// TIA Portal V20 export
FUNCTION_BLOCK "LER_Vision_XGX2000_Conversion"   // FB109, LAD
// stored: Access Published, MemoryReserve 100, SetENOAutomatically false
   VAR_INPUT
      VisionData : "LER_typeVisionMonitoring";
   END_VAR
   VAR_OUTPUT
      VisionDataConvert : "LER_typeVisionResultData";
   END_VAR
BEGIN

REGION Network 1
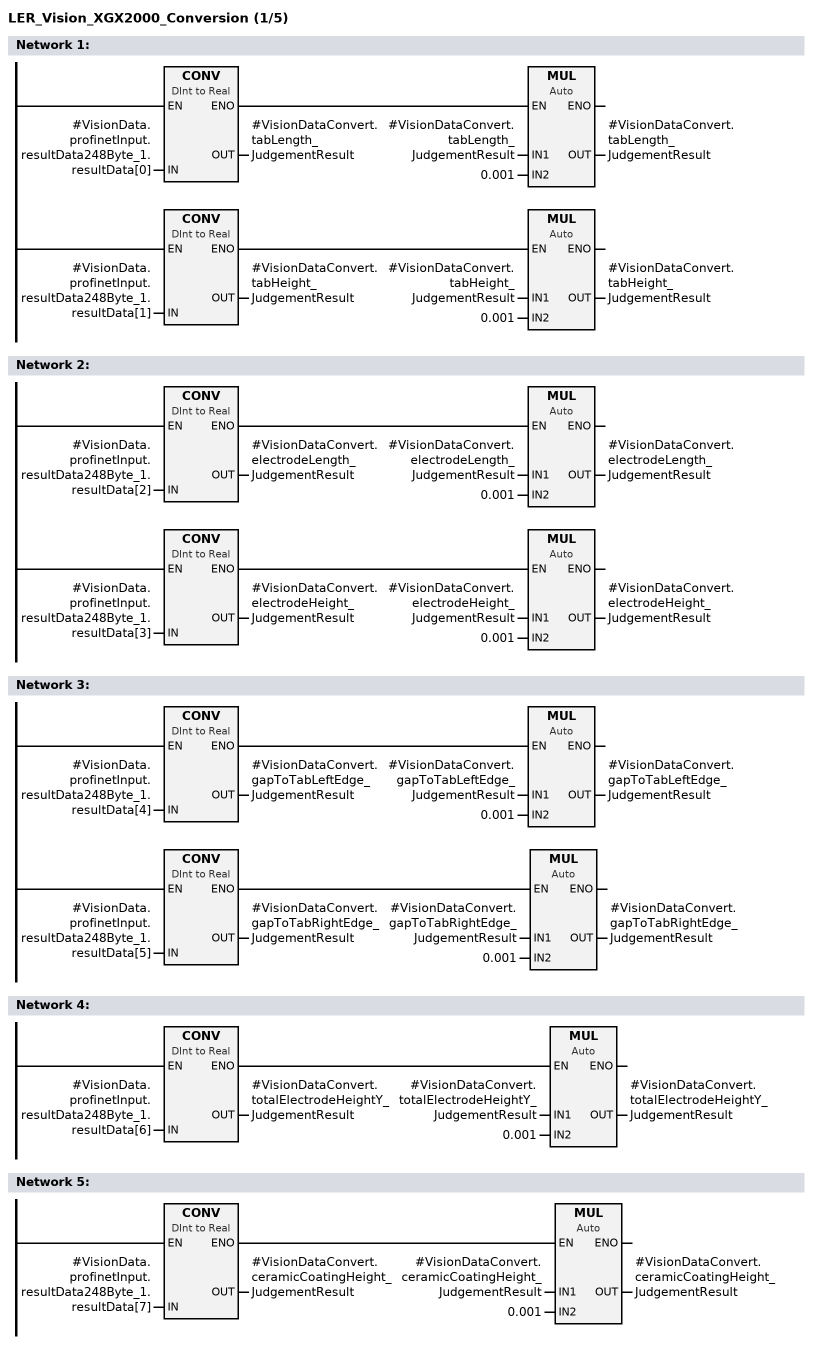
   RUNG wire#powerrail
      { S7_Templates := "[SrcType := DInt, DestType := Real]" } Convert(in := #VisionData.profinetInput.resultData248Byte_1.resultData[0], out => #VisionDataConvert.tabLength_JudgementResult)
      Mul(in1 := #VisionDataConvert.tabLength_JudgementResult, in2 := 0.001, out => #VisionDataConvert.tabLength_JudgementResult)
   END_RUNG
   RUNG wire#powerrail
      { S7_Templates := "[SrcType := DInt, DestType := Real]" } Convert(in := #VisionData.profinetInput.resultData248Byte_1.resultData[1], out => #VisionDataConvert.tabHeight_JudgementResult)
      Mul(in1 := #VisionDataConvert.tabHeight_JudgementResult, in2 := 0.001, out => #VisionDataConvert.tabHeight_JudgementResult)
   END_RUNG
   // the same network as SCL:
   #VisionDataConvert.tabLength_JudgementResult := DINT_TO_REAL(#VisionData.profinetInput.resultData248Byte_1.resultData[0]);
   #VisionDataConvert.tabLength_JudgementResult := #VisionDataConvert.tabLength_JudgementResult * 0.001;
   #VisionDataConvert.tabHeight_JudgementResult := DINT_TO_REAL(#VisionData.profinetInput.resultData248Byte_1.resultData[1]);
   #VisionDataConvert.tabHeight_JudgementResult := #VisionDataConvert.tabHeight_JudgementResult * 0.001;
END_REGION

REGION Network 2
   RUNG wire#powerrail
      { S7_Templates := "[SrcType := DInt, DestType := Real]" } Convert(in := #VisionData.profinetInput.resultData248Byte_1.resultData[2], out => #VisionDataConvert.electrodeLength_JudgementResult)
      Mul(in1 := #VisionDataConvert.electrodeLength_JudgementResult, in2 := 0.001, out => #VisionDataConvert.electrodeLength_JudgementResult)
   END_RUNG
   RUNG wire#powerrail
      { S7_Templates := "[SrcType := DInt, DestType := Real]" } Convert(in := #VisionData.profinetInput.resultData248Byte_1.resultData[3], out => #VisionDataConvert.electrodeHeight_JudgementResult)
      Mul(in1 := #VisionDataConvert.electrodeHeight_JudgementResult, in2 := 0.001, out => #VisionDataConvert.electrodeHeight_JudgementResult)
   END_RUNG
   // the same network as SCL:
   #VisionDataConvert.electrodeLength_JudgementResult := DINT_TO_REAL(#VisionData.profinetInput.resultData248Byte_1.resultData[2]);
   #VisionDataConvert.electrodeLength_JudgementResult := #VisionDataConvert.electrodeLength_JudgementResult * 0.001;
   #VisionDataConvert.electrodeHeight_JudgementResult := DINT_TO_REAL(#VisionData.profinetInput.resultData248Byte_1.resultData[3]);
   #VisionDataConvert.electrodeHeight_JudgementResult := #VisionDataConvert.electrodeHeight_JudgementResult * 0.001;
END_REGION

REGION Network 3
   RUNG wire#powerrail
      { S7_Templates := "[SrcType := DInt, DestType := Real]" } Convert(in := #VisionData.profinetInput.resultData248Byte_1.resultData[4], out => #VisionDataConvert.gapToTabLeftEdge_JudgementResult)
      Mul(in1 := #VisionDataConvert.gapToTabLeftEdge_JudgementResult, in2 := 0.001, out => #VisionDataConvert.gapToTabLeftEdge_JudgementResult)
   END_RUNG
   RUNG wire#powerrail
      { S7_Templates := "[SrcType := DInt, DestType := Real]" } Convert(in := #VisionData.profinetInput.resultData248Byte_1.resultData[5], out => #VisionDataConvert.gapToTabRightEdge_JudgementResult)
      Mul(in1 := #VisionDataConvert.gapToTabRightEdge_JudgementResult, in2 := 0.001, out => #VisionDataConvert.gapToTabRightEdge_JudgementResult)
   END_RUNG
   // the same network as SCL:
   #VisionDataConvert.gapToTabLeftEdge_JudgementResult := DINT_TO_REAL(#VisionData.profinetInput.resultData248Byte_1.resultData[4]);
   #VisionDataConvert.gapToTabLeftEdge_JudgementResult := #VisionDataConvert.gapToTabLeftEdge_JudgementResult * 0.001;
   #VisionDataConvert.gapToTabRightEdge_JudgementResult := DINT_TO_REAL(#VisionData.profinetInput.resultData248Byte_1.resultData[5]);
   #VisionDataConvert.gapToTabRightEdge_JudgementResult := #VisionDataConvert.gapToTabRightEdge_JudgementResult * 0.001;
END_REGION

REGION Network 4
   RUNG wire#powerrail
      { S7_Templates := "[SrcType := DInt, DestType := Real]" } Convert(in := #VisionData.profinetInput.resultData248Byte_1.resultData[6], out => #VisionDataConvert.totalElectrodeHeightY_JudgementResult)
      Mul(in1 := #VisionDataConvert.totalElectrodeHeightY_JudgementResult, in2 := 0.001, out => #VisionDataConvert.totalElectrodeHeightY_JudgementResult)
   END_RUNG
   // the same network as SCL:
   #VisionDataConvert.totalElectrodeHeightY_JudgementResult := DINT_TO_REAL(#VisionData.profinetInput.resultData248Byte_1.resultData[6]);
   #VisionDataConvert.totalElectrodeHeightY_JudgementResult := #VisionDataConvert.totalElectrodeHeightY_JudgementResult * 0.001;
END_REGION

REGION Network 5
   RUNG wire#powerrail
      { S7_Templates := "[SrcType := DInt, DestType := Real]" } Convert(in := #VisionData.profinetInput.resultData248Byte_1.resultData[7], out => #VisionDataConvert.ceramicCoatingHeight_JudgementResult)
      Mul(in1 := #VisionDataConvert.ceramicCoatingHeight_JudgementResult, in2 := 0.001, out => #VisionDataConvert.ceramicCoatingHeight_JudgementResult)
   END_RUNG
   // the same network as SCL:
   #VisionDataConvert.ceramicCoatingHeight_JudgementResult := DINT_TO_REAL(#VisionData.profinetInput.resultData248Byte_1.resultData[7]);
   #VisionDataConvert.ceramicCoatingHeight_JudgementResult := #VisionDataConvert.ceramicCoatingHeight_JudgementResult * 0.001;
END_REGION

REGION Network 6
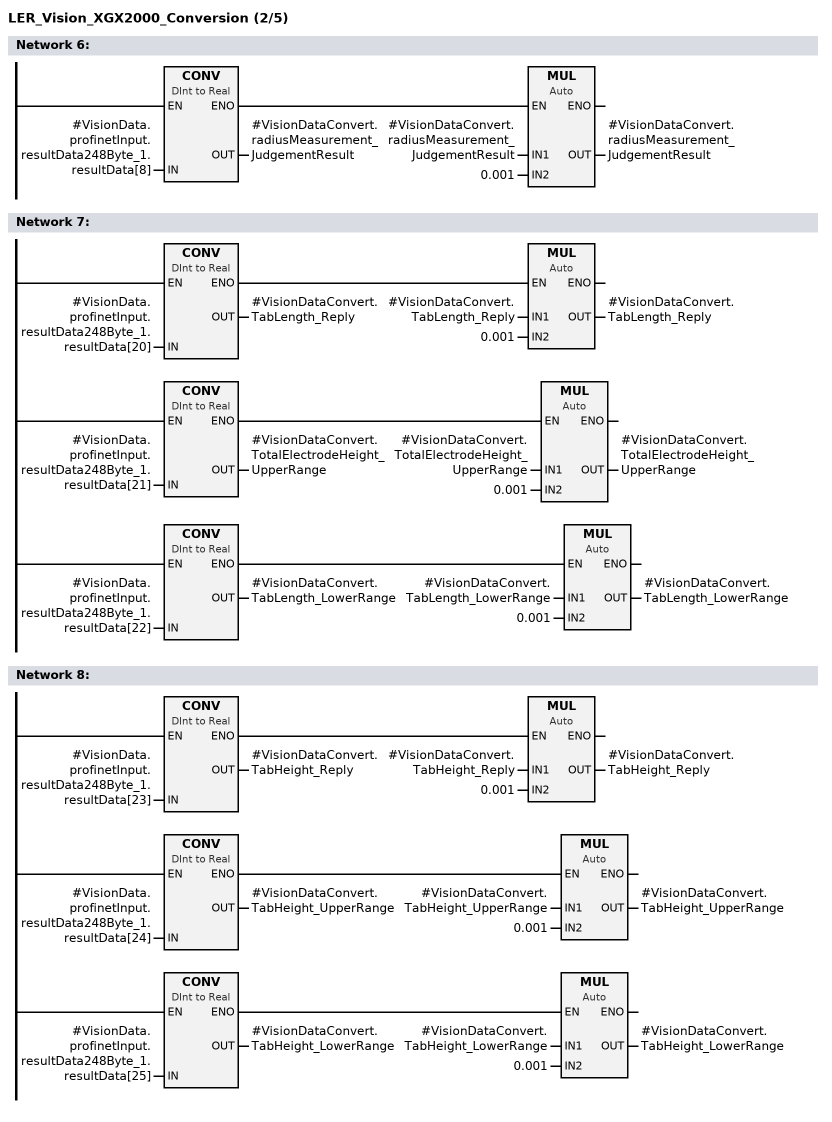
   RUNG wire#powerrail
      { S7_Templates := "[SrcType := DInt, DestType := Real]" } Convert(in := #VisionData.profinetInput.resultData248Byte_1.resultData[8], out => #VisionDataConvert.radiusMeasurement_JudgementResult)
      Mul(in1 := #VisionDataConvert.radiusMeasurement_JudgementResult, in2 := 0.001, out => #VisionDataConvert.radiusMeasurement_JudgementResult)
   END_RUNG
   // the same network as SCL:
   #VisionDataConvert.radiusMeasurement_JudgementResult := DINT_TO_REAL(#VisionData.profinetInput.resultData248Byte_1.resultData[8]);
   #VisionDataConvert.radiusMeasurement_JudgementResult := #VisionDataConvert.radiusMeasurement_JudgementResult * 0.001;
END_REGION

REGION Network 7
   RUNG wire#powerrail
      { S7_Templates := "[SrcType := DInt, DestType := Real]" } Convert(in := #VisionData.profinetInput.resultData248Byte_1.resultData[20], out => #VisionDataConvert.TabLength_Reply)
      Mul(in1 := #VisionDataConvert.TabLength_Reply, in2 := 0.001, out => #VisionDataConvert.TabLength_Reply)
   END_RUNG
   RUNG wire#powerrail
      { S7_Templates := "[SrcType := DInt, DestType := Real]" } Convert(in := #VisionData.profinetInput.resultData248Byte_1.resultData[21], out => #VisionDataConvert.TotalElectrodeHeight_UpperRange)
      Mul(in1 := #VisionDataConvert.TotalElectrodeHeight_UpperRange, in2 := 0.001, out => #VisionDataConvert.TotalElectrodeHeight_UpperRange)
   END_RUNG
   RUNG wire#powerrail
      { S7_Templates := "[SrcType := DInt, DestType := Real]" } Convert(in := #VisionData.profinetInput.resultData248Byte_1.resultData[22], out => #VisionDataConvert.TabLength_LowerRange)
      Mul(in1 := #VisionDataConvert.TabLength_LowerRange, in2 := 0.001, out => #VisionDataConvert.TabLength_LowerRange)
   END_RUNG
   // the same network as SCL:
   #VisionDataConvert.TabLength_Reply := DINT_TO_REAL(#VisionData.profinetInput.resultData248Byte_1.resultData[20]);
   #VisionDataConvert.TabLength_Reply := #VisionDataConvert.TabLength_Reply * 0.001;
   #VisionDataConvert.TotalElectrodeHeight_UpperRange := DINT_TO_REAL(#VisionData.profinetInput.resultData248Byte_1.resultData[21]);
   #VisionDataConvert.TotalElectrodeHeight_UpperRange := #VisionDataConvert.TotalElectrodeHeight_UpperRange * 0.001;
   #VisionDataConvert.TabLength_LowerRange := DINT_TO_REAL(#VisionData.profinetInput.resultData248Byte_1.resultData[22]);
   #VisionDataConvert.TabLength_LowerRange := #VisionDataConvert.TabLength_LowerRange * 0.001;
END_REGION

REGION Network 8
   RUNG wire#powerrail
      { S7_Templates := "[SrcType := DInt, DestType := Real]" } Convert(in := #VisionData.profinetInput.resultData248Byte_1.resultData[23], out => #VisionDataConvert.TabHeight_Reply)
      Mul(in1 := #VisionDataConvert.TabHeight_Reply, in2 := 0.001, out => #VisionDataConvert.TabHeight_Reply)
   END_RUNG
   RUNG wire#powerrail
      { S7_Templates := "[SrcType := DInt, DestType := Real]" } Convert(in := #VisionData.profinetInput.resultData248Byte_1.resultData[24], out => #VisionDataConvert.TabHeight_UpperRange)
      Mul(in1 := #VisionDataConvert.TabHeight_UpperRange, in2 := 0.001, out => #VisionDataConvert.TabHeight_UpperRange)
   END_RUNG
   RUNG wire#powerrail
      { S7_Templates := "[SrcType := DInt, DestType := Real]" } Convert(in := #VisionData.profinetInput.resultData248Byte_1.resultData[25], out => #VisionDataConvert.TabHeight_LowerRange)
      Mul(in1 := #VisionDataConvert.TabHeight_LowerRange, in2 := 0.001, out => #VisionDataConvert.TabHeight_LowerRange)
   END_RUNG
   // the same network as SCL:
   #VisionDataConvert.TabHeight_Reply := DINT_TO_REAL(#VisionData.profinetInput.resultData248Byte_1.resultData[23]);
   #VisionDataConvert.TabHeight_Reply := #VisionDataConvert.TabHeight_Reply * 0.001;
   #VisionDataConvert.TabHeight_UpperRange := DINT_TO_REAL(#VisionData.profinetInput.resultData248Byte_1.resultData[24]);
   #VisionDataConvert.TabHeight_UpperRange := #VisionDataConvert.TabHeight_UpperRange * 0.001;
   #VisionDataConvert.TabHeight_LowerRange := DINT_TO_REAL(#VisionData.profinetInput.resultData248Byte_1.resultData[25]);
   #VisionDataConvert.TabHeight_LowerRange := #VisionDataConvert.TabHeight_LowerRange * 0.001;
END_REGION

REGION Network 9
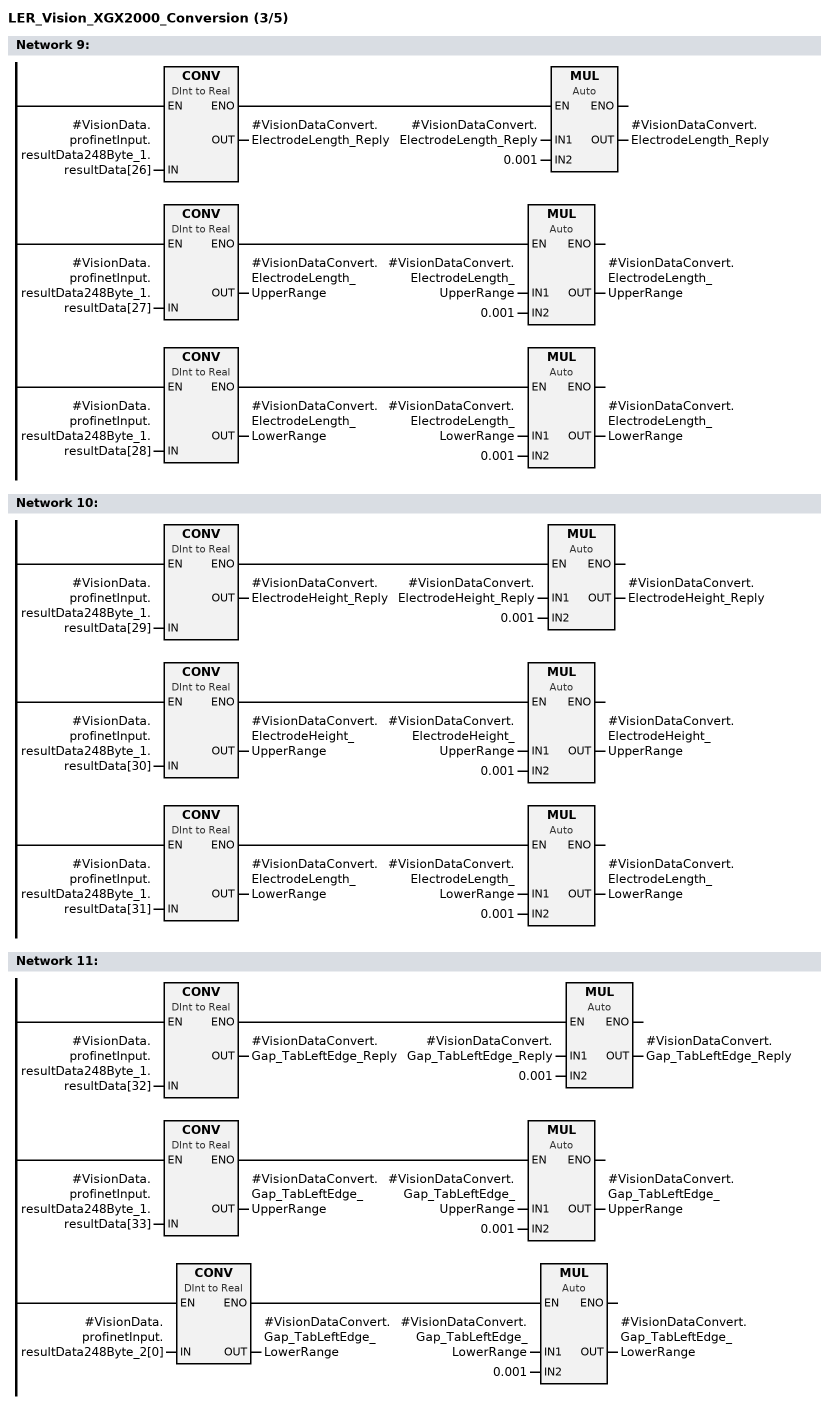
   RUNG wire#powerrail
      { S7_Templates := "[SrcType := DInt, DestType := Real]" } Convert(in := #VisionData.profinetInput.resultData248Byte_1.resultData[26], out => #VisionDataConvert.ElectrodeLength_Reply)
      Mul(in1 := #VisionDataConvert.ElectrodeLength_Reply, in2 := 0.001, out => #VisionDataConvert.ElectrodeLength_Reply)
   END_RUNG
   RUNG wire#powerrail
      { S7_Templates := "[SrcType := DInt, DestType := Real]" } Convert(in := #VisionData.profinetInput.resultData248Byte_1.resultData[27], out => #VisionDataConvert.ElectrodeLength_UpperRange)
      Mul(in1 := #VisionDataConvert.ElectrodeLength_UpperRange, in2 := 0.001, out => #VisionDataConvert.ElectrodeLength_UpperRange)
   END_RUNG
   RUNG wire#powerrail
      { S7_Templates := "[SrcType := DInt, DestType := Real]" } Convert(in := #VisionData.profinetInput.resultData248Byte_1.resultData[28], out => #VisionDataConvert.ElectrodeLength_LowerRange)
      Mul(in1 := #VisionDataConvert.ElectrodeLength_LowerRange, in2 := 0.001, out => #VisionDataConvert.ElectrodeLength_LowerRange)
   END_RUNG
   // the same network as SCL:
   #VisionDataConvert.ElectrodeLength_Reply := DINT_TO_REAL(#VisionData.profinetInput.resultData248Byte_1.resultData[26]);
   #VisionDataConvert.ElectrodeLength_Reply := #VisionDataConvert.ElectrodeLength_Reply * 0.001;
   #VisionDataConvert.ElectrodeLength_UpperRange := DINT_TO_REAL(#VisionData.profinetInput.resultData248Byte_1.resultData[27]);
   #VisionDataConvert.ElectrodeLength_UpperRange := #VisionDataConvert.ElectrodeLength_UpperRange * 0.001;
   #VisionDataConvert.ElectrodeLength_LowerRange := DINT_TO_REAL(#VisionData.profinetInput.resultData248Byte_1.resultData[28]);
   #VisionDataConvert.ElectrodeLength_LowerRange := #VisionDataConvert.ElectrodeLength_LowerRange * 0.001;
END_REGION

REGION Network 10
   RUNG wire#powerrail
      { S7_Templates := "[SrcType := DInt, DestType := Real]" } Convert(in := #VisionData.profinetInput.resultData248Byte_1.resultData[29], out => #VisionDataConvert.ElectrodeHeight_Reply)
      Mul(in1 := #VisionDataConvert.ElectrodeHeight_Reply, in2 := 0.001, out => #VisionDataConvert.ElectrodeHeight_Reply)
   END_RUNG
   RUNG wire#powerrail
      { S7_Templates := "[SrcType := DInt, DestType := Real]" } Convert(in := #VisionData.profinetInput.resultData248Byte_1.resultData[30], out => #VisionDataConvert.ElectrodeHeight_UpperRange)
      Mul(in1 := #VisionDataConvert.ElectrodeHeight_UpperRange, in2 := 0.001, out => #VisionDataConvert.ElectrodeHeight_UpperRange)
   END_RUNG
   RUNG wire#powerrail
      { S7_Templates := "[SrcType := DInt, DestType := Real]" } Convert(in := #VisionData.profinetInput.resultData248Byte_1.resultData[31], out => #VisionDataConvert.ElectrodeLength_LowerRange)
      Mul(in1 := #VisionDataConvert.ElectrodeLength_LowerRange, in2 := 0.001, out => #VisionDataConvert.ElectrodeLength_LowerRange)
   END_RUNG
   // the same network as SCL:
   #VisionDataConvert.ElectrodeHeight_Reply := DINT_TO_REAL(#VisionData.profinetInput.resultData248Byte_1.resultData[29]);
   #VisionDataConvert.ElectrodeHeight_Reply := #VisionDataConvert.ElectrodeHeight_Reply * 0.001;
   #VisionDataConvert.ElectrodeHeight_UpperRange := DINT_TO_REAL(#VisionData.profinetInput.resultData248Byte_1.resultData[30]);
   #VisionDataConvert.ElectrodeHeight_UpperRange := #VisionDataConvert.ElectrodeHeight_UpperRange * 0.001;
   #VisionDataConvert.ElectrodeLength_LowerRange := DINT_TO_REAL(#VisionData.profinetInput.resultData248Byte_1.resultData[31]);
   #VisionDataConvert.ElectrodeLength_LowerRange := #VisionDataConvert.ElectrodeLength_LowerRange * 0.001;
END_REGION

REGION Network 11
   RUNG wire#powerrail
      { S7_Templates := "[SrcType := DInt, DestType := Real]" } Convert(in := #VisionData.profinetInput.resultData248Byte_1.resultData[32], out => #VisionDataConvert.Gap_TabLeftEdge_Reply)
      Mul(in1 := #VisionDataConvert.Gap_TabLeftEdge_Reply, in2 := 0.001, out => #VisionDataConvert.Gap_TabLeftEdge_Reply)
   END_RUNG
   RUNG wire#powerrail
      { S7_Templates := "[SrcType := DInt, DestType := Real]" } Convert(in := #VisionData.profinetInput.resultData248Byte_1.resultData[33], out => #VisionDataConvert.Gap_TabLeftEdge_UpperRange)
      Mul(in1 := #VisionDataConvert.Gap_TabLeftEdge_UpperRange, in2 := 0.001, out => #VisionDataConvert.Gap_TabLeftEdge_UpperRange)
   END_RUNG
   RUNG wire#powerrail
      { S7_Templates := "[SrcType := DInt, DestType := Real]" } Convert(in := #VisionData.profinetInput.resultData248Byte_2[0], out => #VisionDataConvert.Gap_TabLeftEdge_LowerRange)
      Mul(in1 := #VisionDataConvert.Gap_TabLeftEdge_LowerRange, in2 := 0.001, out => #VisionDataConvert.Gap_TabLeftEdge_LowerRange)
   END_RUNG
   // the same network as SCL:
   #VisionDataConvert.Gap_TabLeftEdge_Reply := DINT_TO_REAL(#VisionData.profinetInput.resultData248Byte_1.resultData[32]);
   #VisionDataConvert.Gap_TabLeftEdge_Reply := #VisionDataConvert.Gap_TabLeftEdge_Reply * 0.001;
   #VisionDataConvert.Gap_TabLeftEdge_UpperRange := DINT_TO_REAL(#VisionData.profinetInput.resultData248Byte_1.resultData[33]);
   #VisionDataConvert.Gap_TabLeftEdge_UpperRange := #VisionDataConvert.Gap_TabLeftEdge_UpperRange * 0.001;
   #VisionDataConvert.Gap_TabLeftEdge_LowerRange := DINT_TO_REAL(#VisionData.profinetInput.resultData248Byte_2[0]);
   #VisionDataConvert.Gap_TabLeftEdge_LowerRange := #VisionDataConvert.Gap_TabLeftEdge_LowerRange * 0.001;
END_REGION

REGION Network 12
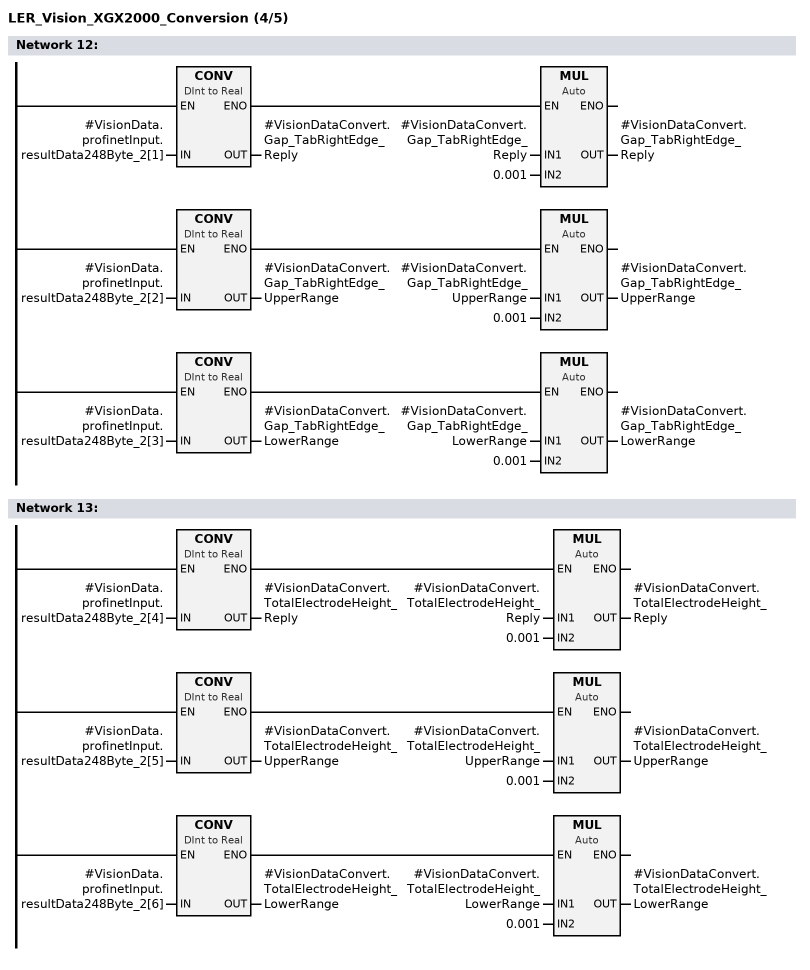
   RUNG wire#powerrail
      { S7_Templates := "[SrcType := DInt, DestType := Real]" } Convert(in := #VisionData.profinetInput.resultData248Byte_2[1], out => #VisionDataConvert.Gap_TabRightEdge_Reply)
      Mul(in1 := #VisionDataConvert.Gap_TabRightEdge_Reply, in2 := 0.001, out => #VisionDataConvert.Gap_TabRightEdge_Reply)
   END_RUNG
   RUNG wire#powerrail
      { S7_Templates := "[SrcType := DInt, DestType := Real]" } Convert(in := #VisionData.profinetInput.resultData248Byte_2[2], out => #VisionDataConvert.Gap_TabRightEdge_UpperRange)
      Mul(in1 := #VisionDataConvert.Gap_TabRightEdge_UpperRange, in2 := 0.001, out => #VisionDataConvert.Gap_TabRightEdge_UpperRange)
   END_RUNG
   RUNG wire#powerrail
      { S7_Templates := "[SrcType := DInt, DestType := Real]" } Convert(in := #VisionData.profinetInput.resultData248Byte_2[3], out => #VisionDataConvert.Gap_TabRightEdge_LowerRange)
      Mul(in1 := #VisionDataConvert.Gap_TabRightEdge_LowerRange, in2 := 0.001, out => #VisionDataConvert.Gap_TabRightEdge_LowerRange)
   END_RUNG
   // the same network as SCL:
   #VisionDataConvert.Gap_TabRightEdge_Reply := DINT_TO_REAL(#VisionData.profinetInput.resultData248Byte_2[1]);
   #VisionDataConvert.Gap_TabRightEdge_Reply := #VisionDataConvert.Gap_TabRightEdge_Reply * 0.001;
   #VisionDataConvert.Gap_TabRightEdge_UpperRange := DINT_TO_REAL(#VisionData.profinetInput.resultData248Byte_2[2]);
   #VisionDataConvert.Gap_TabRightEdge_UpperRange := #VisionDataConvert.Gap_TabRightEdge_UpperRange * 0.001;
   #VisionDataConvert.Gap_TabRightEdge_LowerRange := DINT_TO_REAL(#VisionData.profinetInput.resultData248Byte_2[3]);
   #VisionDataConvert.Gap_TabRightEdge_LowerRange := #VisionDataConvert.Gap_TabRightEdge_LowerRange * 0.001;
END_REGION

REGION Network 13
   RUNG wire#powerrail
      { S7_Templates := "[SrcType := DInt, DestType := Real]" } Convert(in := #VisionData.profinetInput.resultData248Byte_2[4], out => #VisionDataConvert.TotalElectrodeHeight_Reply)
      Mul(in1 := #VisionDataConvert.TotalElectrodeHeight_Reply, in2 := 0.001, out => #VisionDataConvert.TotalElectrodeHeight_Reply)
   END_RUNG
   RUNG wire#powerrail
      { S7_Templates := "[SrcType := DInt, DestType := Real]" } Convert(in := #VisionData.profinetInput.resultData248Byte_2[5], out => #VisionDataConvert.TotalElectrodeHeight_UpperRange)
      Mul(in1 := #VisionDataConvert.TotalElectrodeHeight_UpperRange, in2 := 0.001, out => #VisionDataConvert.TotalElectrodeHeight_UpperRange)
   END_RUNG
   RUNG wire#powerrail
      { S7_Templates := "[SrcType := DInt, DestType := Real]" } Convert(in := #VisionData.profinetInput.resultData248Byte_2[6], out => #VisionDataConvert.TotalElectrodeHeight_LowerRange)
      Mul(in1 := #VisionDataConvert.TotalElectrodeHeight_LowerRange, in2 := 0.001, out => #VisionDataConvert.TotalElectrodeHeight_LowerRange)
   END_RUNG
   // the same network as SCL:
   #VisionDataConvert.TotalElectrodeHeight_Reply := DINT_TO_REAL(#VisionData.profinetInput.resultData248Byte_2[4]);
   #VisionDataConvert.TotalElectrodeHeight_Reply := #VisionDataConvert.TotalElectrodeHeight_Reply * 0.001;
   #VisionDataConvert.TotalElectrodeHeight_UpperRange := DINT_TO_REAL(#VisionData.profinetInput.resultData248Byte_2[5]);
   #VisionDataConvert.TotalElectrodeHeight_UpperRange := #VisionDataConvert.TotalElectrodeHeight_UpperRange * 0.001;
   #VisionDataConvert.TotalElectrodeHeight_LowerRange := DINT_TO_REAL(#VisionData.profinetInput.resultData248Byte_2[6]);
   #VisionDataConvert.TotalElectrodeHeight_LowerRange := #VisionDataConvert.TotalElectrodeHeight_LowerRange * 0.001;
END_REGION

REGION Network 14
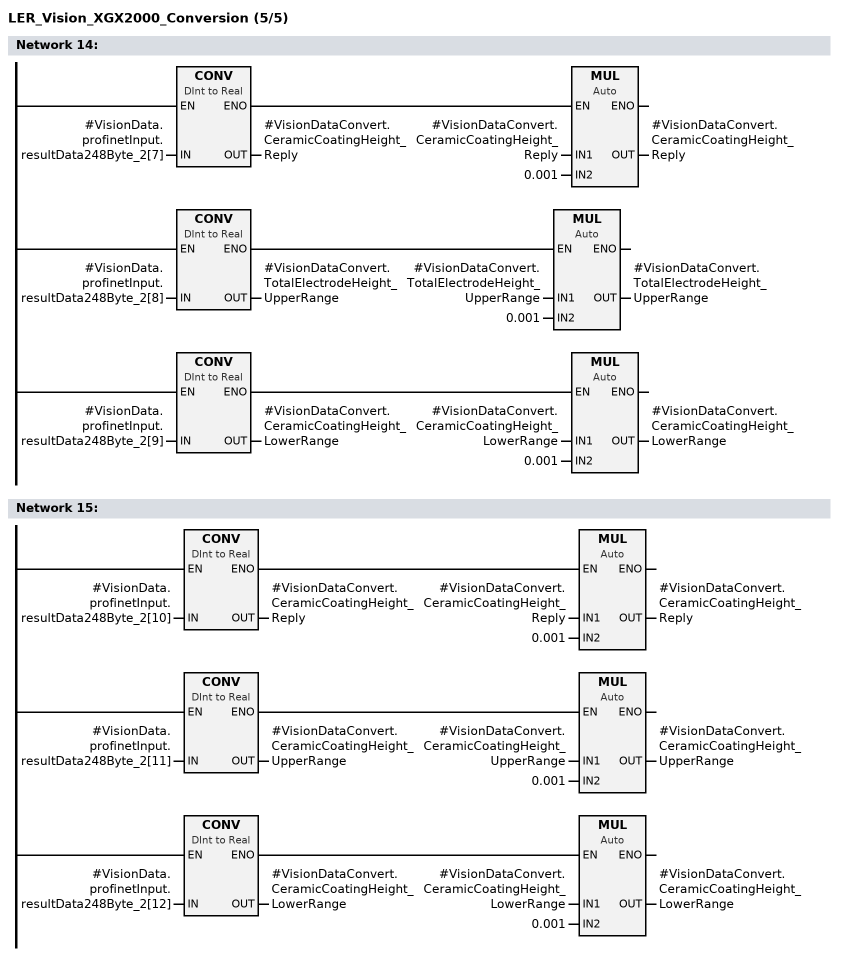
   RUNG wire#powerrail
      { S7_Templates := "[SrcType := DInt, DestType := Real]" } Convert(in := #VisionData.profinetInput.resultData248Byte_2[7], out => #VisionDataConvert.CeramicCoatingHeight_Reply)
      Mul(in1 := #VisionDataConvert.CeramicCoatingHeight_Reply, in2 := 0.001, out => #VisionDataConvert.CeramicCoatingHeight_Reply)
   END_RUNG
   RUNG wire#powerrail
      { S7_Templates := "[SrcType := DInt, DestType := Real]" } Convert(in := #VisionData.profinetInput.resultData248Byte_2[8], out => #VisionDataConvert.TotalElectrodeHeight_UpperRange)
      Mul(in1 := #VisionDataConvert.TotalElectrodeHeight_UpperRange, in2 := 0.001, out => #VisionDataConvert.TotalElectrodeHeight_UpperRange)
   END_RUNG
   RUNG wire#powerrail
      { S7_Templates := "[SrcType := DInt, DestType := Real]" } Convert(in := #VisionData.profinetInput.resultData248Byte_2[9], out => #VisionDataConvert.CeramicCoatingHeight_LowerRange)
      Mul(in1 := #VisionDataConvert.CeramicCoatingHeight_LowerRange, in2 := 0.001, out => #VisionDataConvert.CeramicCoatingHeight_LowerRange)
   END_RUNG
   // the same network as SCL:
   #VisionDataConvert.CeramicCoatingHeight_Reply := DINT_TO_REAL(#VisionData.profinetInput.resultData248Byte_2[7]);
   #VisionDataConvert.CeramicCoatingHeight_Reply := #VisionDataConvert.CeramicCoatingHeight_Reply * 0.001;
   #VisionDataConvert.TotalElectrodeHeight_UpperRange := DINT_TO_REAL(#VisionData.profinetInput.resultData248Byte_2[8]);
   #VisionDataConvert.TotalElectrodeHeight_UpperRange := #VisionDataConvert.TotalElectrodeHeight_UpperRange * 0.001;
   #VisionDataConvert.CeramicCoatingHeight_LowerRange := DINT_TO_REAL(#VisionData.profinetInput.resultData248Byte_2[9]);
   #VisionDataConvert.CeramicCoatingHeight_LowerRange := #VisionDataConvert.CeramicCoatingHeight_LowerRange * 0.001;
END_REGION

REGION Network 15
   RUNG wire#powerrail
      { S7_Templates := "[SrcType := DInt, DestType := Real]" } Convert(in := #VisionData.profinetInput.resultData248Byte_2[10], out => #VisionDataConvert.CeramicCoatingHeight_Reply)
      Mul(in1 := #VisionDataConvert.CeramicCoatingHeight_Reply, in2 := 0.001, out => #VisionDataConvert.CeramicCoatingHeight_Reply)
   END_RUNG
   RUNG wire#powerrail
      { S7_Templates := "[SrcType := DInt, DestType := Real]" } Convert(in := #VisionData.profinetInput.resultData248Byte_2[11], out => #VisionDataConvert.CeramicCoatingHeight_UpperRange)
      Mul(in1 := #VisionDataConvert.CeramicCoatingHeight_UpperRange, in2 := 0.001, out => #VisionDataConvert.CeramicCoatingHeight_UpperRange)
   END_RUNG
   RUNG wire#powerrail
      { S7_Templates := "[SrcType := DInt, DestType := Real]" } Convert(in := #VisionData.profinetInput.resultData248Byte_2[12], out => #VisionDataConvert.CeramicCoatingHeight_LowerRange)
      Mul(in1 := #VisionDataConvert.CeramicCoatingHeight_LowerRange, in2 := 0.001, out => #VisionDataConvert.CeramicCoatingHeight_LowerRange)
   END_RUNG
   // the same network as SCL:
   #VisionDataConvert.CeramicCoatingHeight_Reply := DINT_TO_REAL(#VisionData.profinetInput.resultData248Byte_2[10]);
   #VisionDataConvert.CeramicCoatingHeight_Reply := #VisionDataConvert.CeramicCoatingHeight_Reply * 0.001;
   #VisionDataConvert.CeramicCoatingHeight_UpperRange := DINT_TO_REAL(#VisionData.profinetInput.resultData248Byte_2[11]);
   #VisionDataConvert.CeramicCoatingHeight_UpperRange := #VisionDataConvert.CeramicCoatingHeight_UpperRange * 0.001;
   #VisionDataConvert.CeramicCoatingHeight_LowerRange := DINT_TO_REAL(#VisionData.profinetInput.resultData248Byte_2[12]);
   #VisionDataConvert.CeramicCoatingHeight_LowerRange := #VisionDataConvert.CeramicCoatingHeight_LowerRange * 0.001;
END_REGION
END_FUNCTION_BLOCK
